FUNCTION_BLOCK FbFlush IMPLEMENTS IFlush
VAR_INPUT
END_VAR
VAR_OUTPUT
END_VAR
VAR
END_VAR

{warning 'add method implementation '}
METHOD Flush : BOOL
END_METHOD

{warning 'add property implementation'}
PROPERTY pEndFeedback : BOOL
GET
END_GET
END_PROPERTY

END_FUNCTION_BLOCK

(* stored: Version 1.1.0.1, ProductVersion 3.1.4024.0
   POU FbFlush: Id {0e455ef7-2034-461b-8511-9bfa5fbaa509}, SpecialFunc None
   Method Flush: Id {c4e2aa7e-7e90-4b3f-9194-0a7dad1164cc}
   Property pEndFeedback: Id {a20b3349-1aed-482b-a114-53f06136594e}
   Get Get: Id {288c188e-1c09-4ca2-9362-d33fd687a75b} *)
